	                            #ss_PLCIDTRAYID := CONCAT(IN1 := '0',
	                                                      IN2 := #ss_PLCIDTRAYID);

	                        END_FOR;

	                    END_IF;

	                    // PLCID/TRAYID addition
	                    #ss_PLCIDTRAYID := INSERT(IN1 := #ss_PLCIDTRAYID, IN2 := #is_PLCID_TRAYID, P := 0);

	                    // Delay preparation
	                    #ss_Delay := '';

	                    // Delay integer input conversion to a character string
	                    VAL_STRG(IN := #ii_Delay,
	                             SIZE := 0,
	                             PREC := 0,
	                             FORMAT := 0,
	                             P := 1,
	                             OUT => #ss_Delay);

	                    // Length of the delay character string
	                    #si_DelayLen := LEN(#ss_Delay);

	                    // Delay character string leading zeros addition
	                    IF (#si_DelayLen < 4)
	                    THEN

	                        FOR #si_i := 1 TO 4 - #si_DelayLen DO

	                            #ss_Delay := CONCAT(IN1 := '0',
	                                                IN2 := #ss_Delay);

	                        END_FOR;

	                    END_IF;

	                    // Message preparation

	                    // IDFWD message composing according to the structure: SCN,SCT,RCN,RCT,MT,MSGID,PLCID,DESSYS,DELAY{CRLF}
	                    #ss_Message := CONCAT(IN1 := #iUDT_MsgHeader.SCN,          // Sender IP address
	                                          IN2 := #cc_DL,                        // Comma sign - ","
	                                          IN3 := #iUDT_MsgHeader.SCT,          // Sender Name
	                                          IN4 := #cc_DL,                        // Comma sign - ","
	                                          IN5 := #iUDT_MsgHeader.RCN,          // Receiver IP address
	                                          IN6 := #cc_DL,                        // Comma sign - ","
	                                          IN7 := #iUDT_MsgHeader.RCT,          // Receiver Name
	                                          IN8 := #cc_DL,                        // Comma sign - ","
	                                          IN9 := #cs_IDFWD,                     // Message type - "IDFWD"
	                                          IN10 := #cc_DL,                       // Comma sign - ","
	                                          IN11 := #ss_MSGID,                    // MSGID
	                                          IN12 := #cc_DL,                       // Comma sign - ","
	                                          IN13 := #ss_PLCIDTRAYID,             // PLCID
	                                          IN14 := #cc_DL,                       // Comma sign - ","
	                                          IN15 := #ss_DesSys,                   // Designated system
	                                          IN16 := #cc_DL,                       // Comma sign - ","
	                                          IN17 := #ss_Delay,                    // Delay time
	                                          IN18 := #cs_CRLF);                    // Termination signs - "$R$L"

	                    // Maximum number of the message characters
	                    #si_MaxMsgLen := "FC_GetNrOfArrayEl"(iv_Array := #s_UDT_MessageArray.Character);

	                    // Length of the complete message
	                    #si_MsgLen := LEN(#ss_Message);

	                    // Message array size validation
	                    #ss_Status.InvalidMsgArraySize := #si_MsgLen > #si_MaxMsgLen;

	                    // Message character String conversion into the message array of characters
	                    IF (NOT #ss_Status.InvalidMsgArraySize)
	                    THEN

	                        Strg_TO_Chars(Strg := #ss_Message,
	                                      pChars := 0,
	                                      Cnt => #sui_MsgArrayElNr,
	                                      Chars := #s_UDT_MessageArray.Character);

	                    END_IF;

	                    // Clearing remaining characters in the message character array
	                    IF (NOT #ss_Status.InvalidMsgArraySize)
	                    THEN

	                        // Filling up not used message character array elements with '$00' (ASCII - 16#00)
	                        FILL_BLK(IN := #cc_NULL,
	                                 COUNT := UINT_TO_ULINT(INT_TO_UINT(#si_MaxMsgLen) - #sui_MsgArrayElNr),
	                                 OUT => #s_UDT_MessageArray.Character[#sui_MsgArrayElNr]);

	                    END_IF;

	                    // Message write into a FIFO register
	                    IF (NOT #ss_Status.InvalidMsgArraySize)
	                    THEN

	                        // Mode 'W' - Write FIFO record
	                        "FC_Fifo"(ic_Mode := 'W',
	                                  qUDT_Status => #ss_Status.FIFOStatus,
	                                  qx_Error => #ss_Status.FIFOError,
	                                  qx_Warning => #ss_Status.FIFOWarning,
	                                  iqv_Data := #s_UDT_MessageArray,
	                                  iqUDT_FifoHeader := #iqUDT_FifoHeader,
	                                  iqv_DataBuffer := #iqa_FifoData);

	                        // Message sent as a destination request
	                        "DB_GIN".GIN[#ii_GIN].General.DestReqSend := #ix_DestinationRequest;

	                    END_IF;

	                    // In case of FIFO full, the FIFO full error bit and FIFO collective error bit are set
	                ELSE

	                    #ss_Status.FIFOError := TRUE;
	                    #ss_Status.FIFOStatus.FifoFull := TRUE;

	                END_IF;

	            END_IF;

	        END_REGION

	        REGION 1.4 – Status

	            // Parametrization collective error output
	            #qx_Error :=
	            #ss_Status.InvalidDesSysPar
	            OR #ss_Status.InvalidDelay
	            OR #ss_Status.InvalidGIN
	            OR #ss_Status.InvalidMsgArraySize
	            OR #ss_Status.FIFOError;

	            // Parametrization collective warning output
	            #qx_Warning := #ss_Status.FIFOWarning;

	        END_REGION

	    END_IF;

	END_REGION
END_FUNCTION_BLOCK

FUNCTION_BLOCK "FB_UPSLogon"
TITLE = FB_Logon
{ S7_Optimized_Access := 'TRUE' }
AUTHOR : MHSE
FAMILY : UPS_SpecificCommunication
VERSION : 3.0
// ATTRIBUTES
// AUTO_NUMBER = True
// BLOCK_NUMBER = 57
// END_ATTRIBUTES
//Function block to prepare and send UPS LOGON and FILTER messages.
   VAR_INPUT
      iUDT_Connection { ExternalAccessible := 'False'; ExternalVisible := 'False'; ExternalWritable := 'False'} : "UDT_Connection";   // Connection parameters
      iUDT_MsgHeader { ExternalAccessible := 'False'; ExternalVisible := 'False'; ExternalWritable := 'False'} : "UDT_UPSMessageHeader";   // UPS message header
      ia_MsgType { ExternalAccessible := 'False'; ExternalVisible := 'False'; ExternalWritable := 'False'} : Array[0..34] of String;   // UPS message types
      ix_ConEstablished { ExternalAccessible := 'False'; ExternalVisible := 'False'; ExternalWritable := 'False'} : Bool;   // TCPIP Connection established
   END_VAR

   VAR_OUTPUT
      qx_LogonOk { ExternalAccessible := 'False'; ExternalVisible := 'False'; ExternalWritable := 'False'} : Bool;   // FILTER and LOGON messages sent
   END_VAR

   VAR
      sFB_TSEND {InstructionName := 'TSEND'; LibVersion := '4.0'; ExternalAccessible := 'False'; ExternalVisible := 'False'; ExternalWritable := 'False'; S7_SetPoint := 'False'} : TSEND;   // Siemens "TSEND" block - to send the data over TCPIP socket
      sR_TRIG_ConEstablished {InstructionName := 'R_TRIG'; LibVersion := '1.0'; ExternalAccessible := 'False'; ExternalVisible := 'False'; ExternalWritable := 'False'; S7_SetPoint := 'False'} : R_TRIG;   // Siemens "R_Trig" - to prepare the rising edge trigger on "ix_ConEstablished" signal
      sR_TRIG_SendTrigFilter {InstructionName := 'R_TRIG'; LibVersion := '1.0'; ExternalAccessible := 'False'; ExternalVisible := 'False'; ExternalWritable := 'False'; S7_SetPoint := 'False'} : R_TRIG;   // Siemens "R_Trig" - to prepare the Filter send trigger
      sR_TRIG_SendTrigLogon {InstructionName := 'R_TRIG'; LibVersion := '1.0'; ExternalAccessible := 'False'; ExternalVisible := 'False'; ExternalWritable := 'False'; S7_SetPoint := 'False'} : R_TRIG;   // Siemens "R_Trig" - to prepare the LOGON send trigger
      sa_TSEND { ExternalAccessible := 'False'; ExternalVisible := 'False'; ExternalWritable := 'False'} : Struct   // TSEND block parameter structure
         Status { ExternalAccessible := 'False'; ExternalVisible := 'False'; ExternalWritable := 'False'} : Word;
         Req { ExternalAccessible := 'False'; ExternalVisible := 'False'; ExternalWritable := 'False'} : Bool;
         Busy { ExternalAccessible := 'False'; ExternalVisible := 'False'; ExternalWritable := 'False'} : Bool;
         Done { ExternalAccessible := 'False'; ExternalVisible := 'False'; ExternalWritable := 'False'} : Bool;
         Error { ExternalAccessible := 'False'; ExternalVisible := 'False'; ExternalWritable := 'False'} : Bool;
      END_STRUCT;
      sa_FilterMsg { ExternalAccessible := 'False'; ExternalVisible := 'False'; ExternalWritable := 'False'} : Array[0..699] of Char;   // FILTER message character array
      sa_LogonMsg { ExternalAccessible := 'False'; ExternalVisible := 'False'; ExternalWritable := 'False'} : Array[0..34] of Char;   // LOGON message character array
      ss_Logon { ExternalAccessible := 'False'; ExternalVisible := 'False'; ExternalWritable := 'False'} : String;   // LOGON message character string
      ss_Header { ExternalAccessible := 'False'; ExternalVisible := 'False'; ExternalWritable := 'False'} : String;   // Message header character string
      ss_Filter_1 { ExternalAccessible := 'False'; ExternalVisible := 'False'; ExternalWritable := 'False'} : String;   // FILTER message part 1 character string
      ss_Filter_2 { ExternalAccessible := 'False'; ExternalVisible := 'False'; ExternalWritable := 'False'} : String;   // FILTER message part 2 character string
      ss_Footer { ExternalAccessible := 'False'; ExternalVisible := 'False'; ExternalWritable := 'False'} : String;   // FILTER message footer character string
      sui_ArrayOffset { ExternalAccessible := 'False'; ExternalVisible := 'False'; ExternalWritable := 'False'} : UInt;   // Offset for writing in the array
      sui_FilterArrayElNr { ExternalAccessible := 'False'; ExternalVisible := 'False'; ExternalWritable := 'False'} : UInt;   // Number of written FILTER characters
      sui_LogonArrayElNr { ExternalAccessible := 'False'; ExternalVisible := 'False'; ExternalWritable := 'False'} : UInt;   // Number of written LOGON characters
      si_MaxNrOfMsgTypes { ExternalAccessible := 'False'; ExternalVisible := 'False'; ExternalWritable := 'False'} : Int;   // Maximum number of message types
      si_MaxFilterLen { ExternalAccessible := 'False'; ExternalVisible := 'False'; ExternalWritable := 'False'} : Int;   // Maximum number of FILTER message characters
      si_MaxLogonLen { ExternalAccessible := 'False'; ExternalVisible := 'False'; ExternalWritable := 'False'} : Int;   // Maximum number of LOGON message characters
      si_i { ExternalAccessible := 'False'; ExternalVisible := 'False'; ExternalWritable := 'False'} : Int;   // Loop counter
      sx_LogProc { ExternalAccessible := 'False'; ExternalVisible := 'False'; ExternalWritable := 'False'} : Bool;   // Logon procedure
      sx_FilterSent { ExternalAccessible := 'False'; ExternalVisible := 'False'; ExternalWritable := 'False'} : Bool;   // FILTER message sent
      sx_LogonSent { ExternalAccessible := 'False'; ExternalVisible := 'False'; ExternalWritable := 'False'} : Bool;   // LOGON message sent
   END_VAR

   VAR CONSTANT
      cc_DL : Char := ',';   // Comma sign
      cs_Filter : String := 'FILTER';   // Message type
      cs_Logon : String := 'LOGON';   // Message type
      cs_Pipe : String := ',|,';   // FILTER message element - ,|,
      cs_MT : String := 'MT,$'';   // FILTER message element - MT,'
      cs_Q : String := '$',=';   // FILTER message element - ',=
      cs_CRLF : String := '$R$L';   // Termination signs
   END_VAR


BEGIN
	(*
	----------------------------------------------------------------------------------------

	Version history:
	Date        | Version   | Author        | Remark
	----------------------------------------------------------------------------------------
	24/05/2019  | 0.1       | L.Klar        | first release MHS TIA 15.1
	24/07/2019  | 2.0       | L.Klar        | 2.0 MHS library release TIA 15.1
	23/08/2019  | 2.1       | K.Pokorski    | Comments simplified
	12/11/2019  | 3.0       | P.Majka       | 3.0 MHS library release TIA 15.1
	22/02/2023  | 4.0       | F.Baten       | 4.0 Release TIA 17.5
	*)

	REGION 1 – Connection check

	    // TCIPI connection established rising edge
	    #sR_TRIG_ConEstablished(CLK := #ix_ConEstablished);

	    // Logon process start
	    IF (#sR_TRIG_ConEstablished.Q)                             // Connection established rising edge
	    THEN

	        #sx_LogProc := TRUE;

	    END_IF;

	    // Message send confirmation bits reset in case of connection lost
	    IF (NOT #ix_ConEstablished)                                 // Connection terminated
	    THEN

	        #sx_FilterSent := FALSE;
	        #sx_LogonSent := FALSE;

	    END_IF;

	END_REGION

	REGION 2 – Assembly FILTER message

	    IF (#sx_LogProc)                                            // Logon procedure
	    THEN

	        // Resetting all components of the "Filter" message
	        REGION 2.1 – Initialization

	            #si_i := 0;
	            #sui_ArrayOffset := 0;
	            #sui_FilterArrayElNr := 0;
	            #ss_Header := '';
	            #ss_Filter_1 := '';
	            #ss_Filter_2 := '';
	            #ss_Footer := '';

	        END_REGION

	        REGION 2.2 – Maximum number of the message types array elements

	            #si_MaxNrOfMsgTypes := "FC_GetNrOfArrayEl"(iv_Array := #ia_MsgType);

	        END_REGION

	        REGION 2.3 – Maximum number of the FILTER message array elements

	            #si_MaxFilterLen := "FC_GetNrOfArrayEl"(iv_Array := #sa_FilterMsg);

	        END_REGION

	        // Combining all components of the FILTER message header into one character string
	        REGION 2.4 – Assembly FILTER message header

	            #ss_Header := CONCAT(IN1 := #iUDT_MsgHeader.SCN,       // Sender IP address
	                                 IN2 := #cc_DL,                     // Comma sign - ","
	                                 IN3 := #iUDT_MsgHeader.SCT,       // Sender Name
	                                 IN4 := #cc_DL,                     // Comma sign - ","
	                                 IN5 := #cc_DL,                     // Comma sign - ","
	                                 IN6 := #cc_DL,                     // Comma sign - ","
	                                 IN7 := #cs_Filter,                 // Message type - "FILTER"
	                                 IN8 := #cc_DL);                    // Comma sign - ","

	        END_REGION


	        REGION 2.5 – Assembly FILTER message

	            // Combining all components of the FILTER message into one character string
	            FOR #si_i := 0 TO #si_MaxNrOfMsgTypes - 1 DO

	                IF (#ia_MsgType[#si_i] <> '')       // Message type isn't empty
	                THEN

	                    //  Message charater string conversion to a message array characters
	                    IF (#si_i = 0)                                                          // Loop counter equal to 0
	                    THEN

	                        #ss_Filter_1 := CONCAT(IN1 := #cs_MT,                               // FILTER message constant - "MT,'"
	                                               IN2 := #ia_MsgType[#si_i],                   // Used message type
	                                               IN3 := #cs_Q,                                // FILTER message constant - "',="
	                                               IN4 := #cc_DL);                              // Comma sign - ","

	                        // Message header character string into the character array conversion
	                        Strg_TO_Chars(Strg := #ss_Header,
	                                      pChars := 0,
	                                      Cnt => #sui_ArrayOffset,
	                                      Chars := #sa_FilterMsg);

	                        // FILTER message part 1 character string into the character array conversion
	                        Strg_TO_Chars(Strg := #ss_Filter_1,
	                                      pChars := #sui_ArrayOffset,
	                                      Cnt => #sui_FilterArrayElNr,
	                                      Chars := #sa_FilterMsg);

	                        // Handled message types addition to a filter message
	                    ELSIF (#si_i > 0)                                                       // Loop counter is greater than 0
	                    THEN

	                        #ss_Filter_2 := CONCAT(IN1 := #cs_MT,                               // FILTER message constant - "MT,'"
	                                               IN2 := #ia_MsgType[#si_i],                   // Used message type
	                                               IN3 := #cs_Q,                                // FILTER message constant - "',="
	                                               IN4 := #cs_Pipe);                            // FILTER message constant - ",|,"

	                        // Array offset update
	                        #sui_ArrayOffset += #sui_FilterArrayElNr;

	                        // FILTER message part 2 character string into the character array conversion
	                        Strg_TO_Chars(Strg := #ss_Filter_2,
	                                      pChars := #sui_ArrayOffset,
	                                      Cnt => #sui_FilterArrayElNr,
	                                      Chars := #sa_FilterMsg);

	                    END_IF;

	                    // The message type array element is empty
	                ELSE

	                    EXIT;

	                END_IF;

	            END_FOR;

	        END_REGION

	        REGION 2.6 – Assembly FILTER message footer

	            // FILTER footer creation
	            #ss_Footer := #cs_CRLF;

	            // Array offset update
	            #sui_ArrayOffset += #sui_FilterArrayElNr;

	            // FILTER footer character string into the character array conversion
	            Strg_TO_Chars(Strg := #ss_Footer,
	                          pChars := #sui_ArrayOffset,
	                          Cnt => #sui_FilterArrayElNr,
	                          Chars := #sa_FilterMsg);

	        END_REGION

	        REGION 2.7 – Clearing remaining characters in the message character array

	            // Filling up not used FILTER character array elements with '$00' (ASCII - 16#00)
	            FILL_BLK(IN := '$00',
	                     COUNT := UINT_TO_ULINT(INT_TO_UINT(#si_MaxFilterLen) -
	                                            #sui_FilterArrayElNr -
	                                            #sui_ArrayOffset),
	                     OUT => #sa_FilterMsg[#sui_ArrayOffset + #sui_FilterArrayElNr]);

	        END_REGION

	    END_IF;

	END_REGION

	REGION 3 – Assembly LOGON message

	    IF (#sx_LogProc)        // Logon procedure
	    THEN

	        REGION 3.1 – Initialization

	            #ss_Logon := '';

	        END_REGION

	        REGION 3.2 – Maximum number of the LOGON message array elements

	            #si_MaxLogonLen := "FC_GetNrOfArrayEl"(iv_Array := #sa_LogonMsg);

	        END_REGION

	        REGION 3.3 – Assembly LOGON message

	            #ss_Logon := CONCAT(IN1 := #iUDT_MsgHeader.SCN,        // Sender IP address
	                                IN2 := #cc_DL,                      // Comma sign - ","
	                                IN3 := #iUDT_MsgHeader.SCT,        // Sender Name
	                                IN4 := #cc_DL,                      // Comma sign - ","
	                                IN5 := #cc_DL,                      // Comma sign - ","
	                                IN6 := #cc_DL,                      // Comma sign - ","
	                                IN7 := #cs_Logon,                   // Message type - "LOGON"
	                                IN8 := #cs_CRLF);                   // Termination signs - "$R$L"

	            // LOGON message character string into the character array conversion
	            Strg_TO_Chars(Strg := #ss_Logon,
	                          pChars := 0,
	                          Cnt => #sui_LogonArrayElNr,
	                          Chars := #sa_LogonMsg);

	        END_REGION

	        REGION 3.4 – Clearing remaining characters in the message character array

	            // Filling up not used LOGON character array elements with '$00' (ASCII - 16#00)
	            FILL_BLK(IN := '$00',
	                     COUNT := UINT_TO_ULINT(INT_TO_UINT(#si_MaxLogonLen) -
	                                            #sui_LogonArrayElNr),
	                     OUT => #sa_LogonMsg[#sui_LogonArrayElNr]);

	        END_REGION

	    END_IF;

	END_REGION

	REGION 4 – Send FILTER message

	    REGION 4.1 – Send trigger preparation

	        #sR_TRIG_SendTrigFilter(CLK := NOT #sa_TSEND.#Busy
	                                AND #ix_ConEstablished
	                                AND #sx_LogProc
	                                AND NOT #sx_FilterSent
	                                AND NOT #sx_LogonSent,
	                                Q => #sa_TSEND.#Req);

	    END_REGION

	    REGION 4.2 – Send message

	        IF (NOT #sx_FilterSent               // FILTER message not sent
	            AND NOT #sx_LogonSent)           // LOGON message not sent
	        THEN

	            // FILTER message send
	            #sFB_TSEND(REQ := #sa_TSEND.#Req,
	                       ID := #iUDT_Connection.ID,
	                       LEN := #sui_ArrayOffset + #sui_FilterArrayElNr,
	                       DONE => #sa_TSEND.Done,
	                       BUSY => #sa_TSEND.Busy,
	                       ERROR => #sa_TSEND.Error,
	                       STATUS => #sa_TSEND.Status,
	                       DATA := #sa_FilterMsg);

	            // FILTER sent
	            IF (#sa_TSEND.#Done)        // Operation is done
	            THEN

	                #sx_FilterSent := TRUE;

	            END_IF;

	        END_IF;

	    END_REGION

	END_REGION

	REGION 5 – LOGON message send

	    REGION 5.1 – Send trigger preparation

	        #sR_TRIG_SendTrigLogon(CLK := NOT #sa_TSEND.Busy       // TSEND block not busy
	                               AND #ix_ConEstablished          // Connection established
	                               AND #sx_LogProc                 // Logon procedure
	                               AND #sx_FilterSent              // FILTER message is sent
	                               AND NOT #sx_LogonSent,          // LOGON message is not sent
	                               Q => #sa_TSEND.Req);

	    END_REGION

	    REGION 5.2 – Send message

	        IF (#sx_FilterSent              // FILTER mseesge is sent
	            AND NOT #sx_LogonSent)      // LOGON message is not sent
	        THEN
	            // LOGON message send
	            #sFB_TSEND(REQ := #sa_TSEND.#Req,
	                       ID := #iUDT_Connection.ID,
	                       LEN := #sui_LogonArrayElNr,
	                       DONE => #sa_TSEND.#Done,
	                       BUSY => #sa_TSEND.#Busy,
	                       ERROR => #sa_TSEND.#Error,
	                       STATUS => #sa_TSEND.#Status,
	                       DATA := #sa_LogonMsg);

	            // LOGON sent
	            IF (#sa_TSEND.#Done)        // Operation is done
	            THEN

	                #sx_LogonSent := TRUE;

	            END_IF;

	        END_IF;

	    END_REGION

	END_REGION

	REGION 6 – Reset Logon procedure

	    IF (#sx_FilterSent               // FILTER message sent
	        AND #sx_LogonSent)           // LOGON message sent
	    THEN

	        #sx_LogProc := FALSE;

	    END_IF;

	END_REGION

	REGION 7 – Write outputs

	    #qx_LogonOk :=
	    #sx_FilterSent            // FILTER message sent
	    AND #sx_LogonSent;        // LOGON message sent

	END_REGION
END_FUNCTION_BLOCK

FUNCTION_BLOCK "FB_UPSPLCInfo"
TITLE = FB_PLCInfo
{ S7_Optimized_Access := 'TRUE' }
AUTHOR : MHSE
FAMILY : UPS_SpecificCommunication
VERSION : 3.0
// ATTRIBUTES
// AUTO_NUMBER = True
// BLOCK_NUMBER = 58
// END_ATTRIBUTES
//Function block to prepare and send the UPS PLCINFO message.
   VAR_INPUT
      iUDT_MsgHeader { ExternalAccessible := 'False'; ExternalVisible := 'False'; ExternalWritable := 'False'} : "UDT_UPSMessageHeader";   // UPS message header
      iUDT_MachStat { ExternalAccessible := 'False'; ExternalVisible := 'False'; ExternalWritable := 'False'} : "UDT_UPSMACHSTAT";   // Machine status
      iUDT_ExternalReaders { ExternalAccessible := 'False'; ExternalVisible := 'False'; ExternalWritable := 'False'} : Array[0..15] of "UDT_UPSExternalReader";   // Active camera
      is_ActualDateTime { ExternalAccessible := 'False'; ExternalVisible := 'False'; ExternalWritable := 'False'} : String[23];   // Actual date and time
      is_ModuleName { ExternalAccessible := 'False'; ExternalVisible := 'False'; ExternalWritable := 'False'} : String[2] := 'AB';   // Module type
      is_DeviceNumber { ExternalAccessible := 'False'; ExternalVisible := 'False'; ExternalWritable := 'False'} : String[4] := 'abcd';   // Device number
      iudi_Speed { ExternalAccessible := 'False'; ExternalVisible := 'False'; ExternalWritable := 'False'} : UDInt;   // Conveyor speed [ft/min]
      iudi_SysRevs { ExternalAccessible := 'False'; ExternalVisible := 'False'; ExternalWritable := 'False'} : UDInt;   // Number of system revolutions since sort start
      ii_SendTimeInterval { ExternalAccessible := 'False'; ExternalVisible := 'False'; ExternalWritable := 'False'} : UInt;   // Send time interval [ms]
      ix_ExternalTrigger { ExternalAccessible := 'False'; ExternalVisible := 'False'; ExternalWritable := 'False'} : Bool;   // External trigger to send a message
   END_VAR

   VAR_OUTPUT
      qx_Error { ExternalAccessible := 'False'; ExternalVisible := 'False'; ExternalWritable := 'False'} : Bool;   // Collective error output
      qx_Warning { ExternalAccessible := 'False'; ExternalVisible := 'False'; ExternalWritable := 'False'} : Bool;   // Collective warning output
   END_VAR

   VAR_IN_OUT
      iqUDT_FifoHeader : "UDT_FifoHeader";   // FIFO header
      iqa_FifoData : Array[*] of "UDT_Message";   // FIFO data
      iqdi_UniqueMsgID { ExternalAccessible := 'False'; ExternalVisible := 'False'; ExternalWritable := 'False'} : DInt;   // Unique message ID integer
   END_VAR

   VAR
      sUDT_ActiveCamera { ExternalAccessible := 'False'; ExternalVisible := 'False'; ExternalWritable := 'False'; S7_SetPoint := 'False'} : Array[0..15] of "UDT_UPSExternalReader";   // Active camera status
      sa_MachStatArray { ExternalAccessible := 'False'; ExternalVisible := 'False'; ExternalWritable := 'False'} : Array[0..15] of Byte;   // Machine status array
      sR_TRIG_ExternaReq {InstructionName := 'R_TRIG'; LibVersion := '1.0'; ExternalAccessible := 'False'; ExternalVisible := 'False'; ExternalWritable := 'False'; S7_SetPoint := 'False'} : R_TRIG;   // Siemens "R_TRIG" - to prepare the rising edge trigger on "ix_ExternalTrigger" signal
      sF_TRIG_ExternalReq {InstructionName := 'F_TRIG'; LibVersion := '1.0'; ExternalAccessible := 'False'; ExternalVisible := 'False'; ExternalWritable := 'False'; S7_SetPoint := 'False'} : F_TRIG;   // Siemens "F_TRIG" - to prepare the falling edge trigger on "ix_ExternalTrigger" signal
      sFB_SendPulse { ExternalAccessible := 'False'; ExternalVisible := 'False'; ExternalWritable := 'False'; S7_SetPoint := 'False'} : "FB_Pulse";   // MHS "FB_Pulse" block - to generate preset pulse signal
      sUDT_MessageArray { ExternalAccessible := 'False'; ExternalVisible := 'False'; ExternalWritable := 'False'; S7_SetPoint := 'False'} : "UDT_Message";   // Message character array
      sa_Status { ExternalAccessible := 'False'; ExternalVisible := 'False'; ExternalWritable := 'False'} : Struct   // Status structure
         FIFOStatus { ExternalAccessible := 'False'; ExternalVisible := 'False'; ExternalWritable := 'False'} : "UDT_FifoStatus";   // FIFO status structure
         FIFOError { ExternalAccessible := 'False'; ExternalVisible := 'False'; ExternalWritable := 'False'; S7_SetPoint := 'True'} : Bool;   // FIFO error
         FIFOWarning { ExternalAccessible := 'False'; ExternalVisible := 'False'; ExternalWritable := 'False'; S7_SetPoint := 'True'} : Bool;   // FIFO warning
         InvalidSysRevs { ExternalAccessible := 'False'; ExternalVisible := 'False'; ExternalWritable := 'False'} : Bool;   // Invalid system revolutions number
         InvalidSpeed { ExternalAccessible := 'False'; ExternalVisible := 'False'; ExternalWritable := 'False'} : Bool;   // Invalid conveyor speed
         InvalidMsgArraySize { ExternalAccessible := 'False'; ExternalVisible := 'False'; ExternalWritable := 'False'} : Bool;   // Invalid message array size
      END_STRUCT;
      ss_MsgID { ExternalAccessible := 'False'; ExternalVisible := 'False'; ExternalWritable := 'False'} : String[32];   // Unique message ID
      ss_SysRevs { ExternalAccessible := 'False'; ExternalVisible := 'False'; ExternalWritable := 'False'} : String[4];   // Number of system revolutions since sort start
      ss_Speed { ExternalAccessible := 'False'; ExternalVisible := 'False'; ExternalWritable := 'False'} : String[5];   // Speed
      ss_CameraState { ExternalAccessible := 'False'; ExternalVisible := 'False'; ExternalWritable := 'False'} : String[2];   // Camera state character string
      ss_Header { ExternalAccessible := 'False'; ExternalVisible := 'False'; ExternalWritable := 'False'} : String;   // Header character string
      ss_Message { ExternalAccessible := 'False'; ExternalVisible := 'False'; ExternalWritable := 'False'} : String;   // Message character string
      ss_ActiveCamera { ExternalAccessible := 'False'; ExternalVisible := 'False'; ExternalWritable := 'False'} : String;   // Active camera character string
      ss_MachStat { ExternalAccessible := 'False'; ExternalVisible := 'False'; ExternalWritable := 'False'} : String;   // Machine status character string
      ss_MachStatPart { ExternalAccessible := 'False'; ExternalVisible := 'False'; ExternalWritable := 'False'} : String;   // Part of the machine status character string
      sui_MsgArrayElNr { ExternalAccessible := 'False'; ExternalVisible := 'False'; ExternalWritable := 'False'} : UInt;   // Number of written message characters
      sui_ArrayOffset { ExternalAccessible := 'False'; ExternalVisible := 'False'; ExternalWritable := 'False'} : UInt;   // Offset for writing in the array
      si_MaxMsgLen { ExternalAccessible := 'False'; ExternalVisible := 'False'; ExternalWritable := 'False'} : Int;   // Maximum message length
      si_MsgLen { ExternalAccessible := 'False'; ExternalVisible := 'False'; ExternalWritable := 'False'} : Int;   // Message character string length
      si_SysRevsLen { ExternalAccessible := 'False'; ExternalVisible := 'False'; ExternalWritable := 'False'} : Int;   // System revolutions character string length
      si_i { ExternalAccessible := 'False'; ExternalVisible := 'False'; ExternalWritable := 'False'} : Int;   // Loop counter
      sx_NewCameraState { ExternalAccessible := 'False'; ExternalVisible := 'False'; ExternalWritable := 'False'} : Bool;   // Camera state changed
   END_VAR

   VAR CONSTANT
      cc_NULL : Char := '$00';   // NULL sign
      cc_Dash : Char := '-';   // Dash sign
      cc_DL : Char := ',';   // Comma sign
      cs_CamOn : String := '|1';   // Camera state - True
      cs_CamOff : String := '|0';   // Camera state - False
      cs_PLCInfo : String := 'PLCINFO';   // Message type
      cs_CRLF : String := '$R$L';   // Termination signs
   END_VAR


BEGIN
	(*
	----------------------------------------------------------------------------------------

	Version history:
	Date        | Version   | Author        | Remark
	----------------------------------------------------------------------------------------
	24/05/2019  | 0.1       | L.Klar        | first release MHS TIA 15.1
	13/06/2019  | 0.2       | A.Nowak       | Replacement of instruction if for direct write into variable - Region 2 and 3 and 4.10
	28/06/2019  | 0.4       | A.Nowak       | Changing conditions for error occuring and status update
	18/07/2019  | 0.5       | L.Klar        | Status handling changed
	24/07/2019  | 2.0       | L.Klar        | 2.0 MHS library release TIA 15.1
	19/08/2019  | 2.1       | L.Klar        | Cyclic and event message handling added
	23/08/2019  | 2.2       | K.Pokorski    | Bool to byte block changed to direct reference, comments simplified
	20/09/2019  | 2.3       | M.Kurpiers    | Change - status to struct
	01/10/2019  | 2.4       | A.Nowak       | Implementation of the new FIFO block
	12/11/2019  | 3.0       | P.Majka       | 3.0 MHS library release TIA 15.1
	22/02/2023  | 4.0       | F.Baten       | 4.0 Release TIA 17.5
	02/05/2024  | 4.1       | J.Majer      | Datatype conversions changed from automatic to explicit, to accomodate IEC 61131-3 standard
	*)

	REGION 1 – Message send trigger

	    // Custom pulse to create cyclic trigger
	    #sFB_SendPulse(iudi_PulseTime := #ii_SendTimeInterval);

	    // Camera state check
	    #sx_NewCameraState := #sUDT_ActiveCamera <> #iUDT_ExternalReaders;
	    #sUDT_ActiveCamera := #iUDT_ExternalReaders;                             // Move new camera state to block memory

	    // Preparation of the rising and falling edge on the external request to send signal
	    #sR_TRIG_ExternaReq(CLK := #ix_ExternalTrigger);
	    #sF_TRIG_ExternalReq(CLK := #ix_ExternalTrigger);

	END_REGION

	REGION 2 – PLCInfo message request

	    // Condition of sending the message
	    IF (#sFB_SendPulse.qx_Pulse                // Cyclic trigger
	        OR #sx_NewCameraState                   // Camera state changed
	        OR #sR_TRIG_ExternaReq.Q               // External trigger rising edge
	        OR #sF_TRIG_ExternalReq.Q)             // External trigger falling edge
	    THEN

	        REGION 2.1 – FIFO header status update

	            // Mode 'S' - FIFO register status update
	            "FC_Fifo"(ic_Mode := 'S',
	                      qUDT_Status => #sa_Status.FIFOStatus,
	                      qx_Error => #sa_Status.FIFOError,
	                      qx_Warning => #sa_Status.FIFOWarning,
	                      iqv_Data := #sUDT_MessageArray,
	                      iqUDT_FifoHeader := #iqUDT_FifoHeader,
	                      iqv_DataBuffer := #iqa_FifoData);


	        END_REGION

	        REGION 2.2 – Conveyor speed validation

	            #sa_Status.InvalidSpeed :=
	            #iudi_Speed < 0
	            OR #iudi_Speed > 99999;

	        END_REGION

	        REGION 2.3 – System revolutions number validation

	            #sa_Status.InvalidSysRevs :=
	            #iudi_SysRevs < 0
	            OR #iudi_SysRevs > 9999;

	        END_REGION

	        REGION 2.4 – PLCINFO message preparation

	            IF (NOT #sa_Status.InvalidSysRevs                                // System revolutions number is valid
	                AND NOT #sa_Status.InvalidSpeed                              // Conveyor speed is valid
	                AND NOT #sa_Status.FIFOError)                                // No FIFO errors
	            THEN

	                IF (NOT #iqUDT_FifoHeader.Status.Full)                      // FIFO isn't full
	                THEN

	                    // Unique MSGID
	                    "FC_UPSMsgId"(is_ActualDateTime := #is_ActualDateTime,
	                                  is_ModuleName := #is_ModuleName,
	                                  is_DeviceNumber := #is_DeviceNumber,
	                                  iqs_MSGID := #ss_MsgID,
	                                  iqdi_UniqueMsgID := #iqdi_UniqueMsgID);


	                    // Conveyor speed conversion
	                    VAL_STRG(IN := #iudi_Speed,
	                             SIZE := 0,
	                             PREC := 0,
	                             FORMAT := 0,
	                             P := 1,
	                             OUT => #ss_Speed);

	                    // Machine status conversion
	                    #sa_MachStatArray[0].%X0 := #iUDT_MachStat."OpsNormal".StopMCP;                     // MCP Stop PB          // Byte 1, Bit 0 - Operator Stop MCP Panel
	                    #sa_MachStatArray[0].%X1 := #iUDT_MachStat."OpsNormal".StopRemoteCon1;              // SSP         // Byte 1, Bit 1 - Operator Stop Remote Console 1
	                    #sa_MachStatArray[0].%X2 := #iUDT_MachStat."OpsNormal".StopRemoteCon2;              // SSP         // Byte 1, Bit 2 - Operator Stop Remote Console 2
	                    #sa_MachStatArray[0].%X3 := #iUDT_MachStat."OpsNormal".BuildingStop;                // MCP Estop         // Byte 1, Bit 3 - Building Stop via HMI
	                    #sa_MachStatArray[0].%X4 := #iUDT_MachStat."OpsNormal".BuildingBreak;               // false         // Byte 1, Bit 4 - Building Break Time via HMI
	                    #sa_MachStatArray[0].%X5 := #iUDT_MachStat."OpsNormal".PowerSaveShutdown;           // system energy save       // Byte 1, Bit 5 - Power Save Shutdown
	                    #sa_MachStatArray[0].%X6 := #iUDT_MachStat."OpsNormal".SorterNotAtSpeed;            //False        // Byte 1, Bit 6 - Sorter Not at speed
	                    #sa_MachStatArray[0].%X7 := #iUDT_MachStat."OpsNormal".MaintenanceSysMode;          // Manual      // Byte 1, Bit 7 - System in Maintenance Mode

	                    #sa_MachStatArray[1].%X0 := #iUDT_MachStat."OpsNormal".Spare_8;                     // Byte 2, Bit 0 - Future / or Machine Specific (To be identified)
	                    #sa_MachStatArray[1].%X1 := #iUDT_MachStat."OpsNormal".Spare_9;                     // Byte 2, Bit 1 - Future / or Machine Specific (To be identified)
	                    #sa_MachStatArray[1].%X2 := #iUDT_MachStat."OpsNormal".Spare_10;                    // Byte 2, Bit 2 - Future / or Machine Specific (To be identified)
	                    #sa_MachStatArray[1].%X3 := #iUDT_MachStat."OpsNormal".Spare_11;                    // Byte 2, Bit 3 - Future / or Machine Specific (To be identified)
	                    #sa_MachStatArray[1].%X4 := #iUDT_MachStat."OpsNormal".Spare_12;                    // Byte 2, Bit 4 - Future / or Machine Specific (To be identified)
	                    #sa_MachStatArray[1].%X5 := #iUDT_MachStat."OpsNormal".Spare_13;                    // Byte 2, Bit 5 - Future / or Machine Specific (To be identified)
	                    #sa_MachStatArray[1].%X6 := #iUDT_MachStat."OpsNormal".Spare_14;                    // Byte 2, Bit 6 - Future / or Machine Specific (To be identified)
	                    #sa_MachStatArray[1].%X7 := #iUDT_MachStat."OpsNormal".Spare_15;                    // Byte 2, Bit 7 - Future / or Machine Specific (To be identified)


	                    #sa_MachStatArray[2].%X0 := #iUDT_MachStat."OpsNormal".Spare_16;                    // Byte 3, Bit 0 - Future / or Machine Specific (To be identified)
	                    #sa_MachStatArray[2].%X1 := #iUDT_MachStat."OpsNormal".Spare_17;                    // Byte 3, Bit 1 - Future / or Machine Specific (To be identified)
	                    #sa_MachStatArray[2].%X2 := #iUDT_MachStat."OpsNormal".Spare_18;                    // Byte 3, Bit 2 - Future / or Machine Specific (To be identified)
	                    #sa_MachStatArray[2].%X3 := #iUDT_MachStat."OpsNormal".Spare_19;                    // Byte 3, Bit 3 - Future / or Machine Specific (To be identified)
	                    #sa_MachStatArray[2].%X4 := #iUDT_MachStat."OpsNormal".Spare_20;                    // Byte 3, Bit 4 - Future / or Machine Specific (To be identified)
	                    #sa_MachStatArray[2].%X5 := #iUDT_MachStat."OpsNormal".Spare_21;                    // Byte 3, Bit 5 - Future / or Machine Specific (To be identified)
	                    #sa_MachStatArray[2].%X6 := #iUDT_MachStat."OpsNormal".Spare_22;                    // Byte 3, Bit 6 - Future / or Machine Specific (To be identified)
	                    #sa_MachStatArray[2].%X7 := #iUDT_MachStat."OpsNormal".Spare_23;                    // Byte 3, Bit 7 - Future / or Machine Specific (To be identified)


	                    #sa_MachStatArray[3].%X0 := #iUDT_MachStat."OpsNormal".Spare_24;                    // Byte 4, Bit 0 - Future / or Machine Specific (To be identified)
	                    #sa_MachStatArray[3].%X1 := #iUDT_MachStat."OpsNormal".Spare_25;                    // Byte 4, Bit 1 - Future / or Machine Specific (To be identified)
	                    #sa_MachStatArray[3].%X2 := #iUDT_MachStat."OpsNormal".Spare_26;                    // Byte 4, Bit 2 - Future / or Machine Specific (To be identified)
	                    #sa_MachStatArray[3].%X3 := #iUDT_MachStat."OpsNormal".Spare_27;                    // Byte 4, Bit 3 - Future / or Machine Specific (To be identified)
	                    #sa_MachStatArray[3].%X4 := #iUDT_MachStat."OpsNormal".Spare_28;                    // Byte 4, Bit 4 - Future / or Machine Specific (To be identified)
	                    #sa_MachStatArray[3].%X5 := #iUDT_MachStat."OpsNormal".Spare_29;                    // Byte 4, Bit 5 - Future / or Machine Specific (To be identified)
	                    #sa_MachStatArray[3].%X6 := #iUDT_MachStat."OpsNormal".Spare_30;                    // Byte 4, Bit 6 - Future / or Machine Specific (To be identified)
	                    #sa_MachStatArray[3].%X7 := #iUDT_MachStat."OpsNormal".Spare_31;                    // Byte 4, Bit 7 - Future / or Machine Specific (To be identified)


	                    #sa_MachStatArray[4].%X0 := #iUDT_MachStat.SafetyFaults.BuildingEStop;              // comm false           // Byte 5, Bit 0 - Building Emergency Stop
	                    #sa_MachStatArray[4].%X1 := #iUDT_MachStat.SafetyFaults.SystemEStop;                // MCP Estop          // Byte 5, Bit 1 - System Emergency Stop
	                    #sa_MachStatArray[4].%X2 := #iUDT_MachStat.SafetyFaults.EmerPullCord;               // Byte 5, Bit 2 - Emergency Pull Cord
	                    #sa_MachStatArray[4].%X3 := #iUDT_MachStat.SafetyFaults.PhotoEyeBlock1;             // Byte 5, Bit 3 - Safety Photo Eye Blocked (Long Range Photo Eye) 1
	                    #sa_MachStatArray[4].%X4 := #iUDT_MachStat.SafetyFaults.PlatformLockout1;           // Byte 5, Bit 4 - Platform Lockout 1
	                    #sa_MachStatArray[4].%X5 := #iUDT_MachStat.SafetyFaults.PlatformLockout2;           // Byte 5, Bit 5 - Platform Lockout 2
	                    #sa_MachStatArray[4].%X6 := #iUDT_MachStat.SafetyFaults.PhotoEyeBlock2;             // Byte 5, Bit 6 - Safety Photo Eye Blocked (Long Range Photo Eye) 2
	                    #sa_MachStatArray[4].%X7 := #iUDT_MachStat.SafetyFaults.PhotoEyeBlock3;             // Byte 5, Bit 7 - Safety Photo Eye Blocked (Long Range Photo Eye) 3


	                    #sa_MachStatArray[5].%X0 := #iUDT_MachStat.SafetyFaults.Spare_8;                    // Byte 6, Bit 0 - Future / or Machine Specific (To be identified)
	                    #sa_MachStatArray[5].%X1 := #iUDT_MachStat.SafetyFaults.Spare_9;                    // Byte 6, Bit 1 - Future / OR Machine Specific (TO be identified)
	                    #sa_MachStatArray[5].%X2 := #iUDT_MachStat.SafetyFaults.Spare_10;                   // Byte 6, Bit 2 - Future / or Machine Specific (To be identified)
	                    #sa_MachStatArray[5].%X3 := #iUDT_MachStat.SafetyFaults.Spare_11;                   // Byte 6, Bit 3 - Future / or Machine Specific (To be identified)
	                    #sa_MachStatArray[5].%X4 := #iUDT_MachStat.SafetyFaults.Spare_12;                   // Byte 6, Bit 4 - Future / or Machine Specific (To be identified)
	                    #sa_MachStatArray[5].%X5 := #iUDT_MachStat.SafetyFaults.Spare_13;                   // Byte 6, Bit 5 - Future / or Machine Specific (To be identified)
	                    #sa_MachStatArray[5].%X6 := #iUDT_MachStat.SafetyFaults.Spare_14;                   // Byte 6, Bit 6 - Future / or Machine Specific (To be identified)
	                    #sa_MachStatArray[5].%X7 := #iUDT_MachStat.SafetyFaults.Spare_15;                   // Byte 6, Bit 7 - Future / or Machine Specific (To be identified)


	                    #sa_MachStatArray[6].%X0 := #iUDT_MachStat.SafetyFaults.Spare_16;                   // Byte 7, Bit 0 - Future / or Machine Specific (To be identified)
	                    #sa_MachStatArray[6].%X1 := #iUDT_MachStat.SafetyFaults.Spare_17;                   // Byte 7, Bit 1 - Future / or Machine Specific (To be identified)
	                    #sa_MachStatArray[6].%X2 := #iUDT_MachStat.SafetyFaults.Spare_18;                   // Byte 7, Bit 2 - Future / or Machine Specific (To be identified)
	                    #sa_MachStatArray[6].%X3 := #iUDT_MachStat.SafetyFaults.Spare_19;                   // Byte 7, Bit 3 - Future / or Machine Specific (To be identified)
	                    #sa_MachStatArray[6].%X4 := #iUDT_MachStat.SafetyFaults.Spare_20;                   // Byte 7, Bit 4 - Future / or Machine Specific (To be identified)
	                    #sa_MachStatArray[6].%X5 := #iUDT_MachStat.SafetyFaults.Spare_21;                   // Byte 7, Bit 5 - Future / or Machine Specific (To be identified)
	                    #sa_MachStatArray[6].%X6 := #iUDT_MachStat.SafetyFaults.Spare_22;                   // Byte 7, Bit 6 - Future / or Machine Specific (To be identified)
	                    #sa_MachStatArray[6].%X7 := #iUDT_MachStat.SafetyFaults.Spare_23;                   // Byte 7, Bit 7 - Future / or Machine Specific (To be identified)


	                    #sa_MachStatArray[7].%X0 := #iUDT_MachStat.SafetyFaults.Spare_24;                   // Byte 8, Bit 0 - Future / or Machine Specific (To be identified)
	                    #sa_MachStatArray[7].%X1 := #iUDT_MachStat.SafetyFaults.Spare_25;                   // Byte 8, Bit 1 - Future / or Machine Specific (To be identified)
	                    #sa_MachStatArray[7].%X2 := #iUDT_MachStat.SafetyFaults.Spare_26;                   // Byte 8, Bit 2 - Future / or Machine Specific (To be identified)
	                    #sa_MachStatArray[7].%X3 := #iUDT_MachStat.SafetyFaults.Spare_27;                   // Byte 8, Bit 3 - Future / or Machine Specific (To be identified)
	                    #sa_MachStatArray[7].%X4 := #iUDT_MachStat.SafetyFaults.Spare_28;                   // Byte 8, Bit 4 - Future / or Machine Specific (To be identified)
	                    #sa_MachStatArray[7].%X5 := #iUDT_MachStat.SafetyFaults.Spare_29;                   // Byte 8, Bit 5 - Future / or Machine Specific (To be identified)
	                    #sa_MachStatArray[7].%X6 := #iUDT_MachStat.SafetyFaults.Spare_30;                   // Byte 8, Bit 6 - Future / or Machine Specific (To be identified)
	                    #sa_MachStatArray[7].%X7 := #iUDT_MachStat.SafetyFaults.Spare_31;                   // Byte 8, Bit 7 - Future / or Machine Specific (To be identified)


	                    #sa_MachStatArray[8].%X0 := #iUDT_MachStat.SystemFaults.PLCRackFault;               // RIO Error     // Byte 9, Bit 0 - PLC Rack Fault
	                    #sa_MachStatArray[8].%X1 := #iUDT_MachStat.SystemFaults.EncoderFault;               // Byte 9, Bit 1 - Encoder Fault
	                    #sa_MachStatArray[8].%X2 := #iUDT_MachStat.SystemFaults.TipperOrDiverterFault;      // Byte 9, Bit 2 - Tipper / Diverter Fault
	                    #sa_MachStatArray[8].%X3 := #iUDT_MachStat.SystemFaults.TCPConFail;                 // Byte 9, Bit 3 - TCP Connection Failure
	                    #sa_MachStatArray[8].%X4 := #iUDT_MachStat.SystemFaults.SensorJam;                  // Byte 9, Bit 4 - Package Detect Sensor Jam
	                    #sa_MachStatArray[8].%X5 := #iUDT_MachStat.SystemFaults.CamOrScanFail;              // health        // Byte 9, Bit 5 - Camera / Scanner Failure
	                    #sa_MachStatArray[8].%X6 := #iUDT_MachStat.SystemFaults.InductPEJam;                // Byte 9, Bit 6 - Induct Photo Eye Jam
	                    #sa_MachStatArray[8].%X7 := #iUDT_MachStat.SystemFaults.SortVerificationPEJam;      // Byte 9, Bit 7 - Sort Verification Photo Eye Jam


	                    #sa_MachStatArray[9].%X0 := #iUDT_MachStat.SystemFaults.TakeAwayConvPEJam;          // Byte 10, Bit 0 - Take Away Conveyor Photo Eye Jam
	                    #sa_MachStatArray[9].%X1 := #iUDT_MachStat.SystemFaults.SorterMechFault;            // Byte 10, Bit 1 - Sorter Mechanical Fault
	                    #sa_MachStatArray[9].%X2 := #iUDT_MachStat.SystemFaults.Spare_10;                   // Byte 10, Bit 2 - Future / or Machine Specific (To be identified)
	                    #sa_MachStatArray[9].%X3 := #iUDT_MachStat.SystemFaults.SorterJam;                  // Byte 10, Bit 3 - Sorter Jam (Logical Failure)
	                    #sa_MachStatArray[9].%X4 := #iUDT_MachStat.SystemFaults.InductPCAlignmentError;     // Byte 10, Bit 4 - Induct Photo Cell Alignment Error
	                    #sa_MachStatArray[9].%X5 := #iUDT_MachStat.SystemFaults.MotorFault;                 // Byte 10, Bit 5 - Motor Fault
	                    #sa_MachStatArray[9].%X6 := #iUDT_MachStat.SystemFaults.PowerFault;                 // PDP                // Byte 10, Bit 6 - Power Fault
	                    #sa_MachStatArray[9].%X7 := #iUDT_MachStat.SystemFaults.Spare_15;                   // Byte 10, Bit 7 - Future / or Machine Specific (To be identified)


	                    #sa_MachStatArray[10].%X0 := #iUDT_MachStat.SystemFaults.IOComError;                // Byte 11, Bit 0 - I/O Communications Error
	                    #sa_MachStatArray[10].%X1 := #iUDT_MachStat.SystemFaults.RemoteIOComError;          // Byte 11, Bit 1 - Remote I/O Communications Error
	                    #sa_MachStatArray[10].%X2 := #iUDT_MachStat.SystemFaults.XLeChatComError;           // Byte 11, Bit 2 - XLe chat Communications Error
	                    #sa_MachStatArray[10].%X3 := #iUDT_MachStat.SystemFaults.SerialComError;            // Byte 11, Bit 3 - Serial Communications Error
	                    #sa_MachStatArray[10].%X4 := #iUDT_MachStat.SystemFaults.SubsystemError;            // camera error           // Byte 11, Bit 4 - Subsystem Error (Scale, Camera, etc…)
	                    #sa_MachStatArray[10].%X5 := #iUDT_MachStat.SystemFaults.VDFFault;                  // Byte 11, Bit 5 - VDF Fault
	                    #sa_MachStatArray[10].%X6 := #iUDT_MachStat.SystemFaults.SystemResetInitiated;      // Byte 11, Bit 6 - System Reset Initiated
	                    #sa_MachStatArray[10].%X7 := #iUDT_MachStat.SystemFaults.PFCStopMode;               // Byte 11, Bit 7 - PFC not in Run Mode


	                    #sa_MachStatArray[11].%X0 := #iUDT_MachStat.SystemFaults.NoHitPoints;               // Byte 12, Bit 0 - No Hit points / Divert Set Points found
	                    #sa_MachStatArray[11].%X1 := #iUDT_MachStat.SystemFaults.MissingTraysDetected;      // Byte 12, Bit 1 - Missing Trays Detected
	                    #sa_MachStatArray[11].%X2 := #iUDT_MachStat.SystemFaults.DataFault;                 // Byte 12, Bit 2 - Data Fault, X number of sequential missing valid SORT messages
	                    #sa_MachStatArray[11].%X3 := #iUDT_MachStat.SystemFaults.Spare_27;                  // Byte 12, Bit 3 - Future / or Machine Specific (To be identified)
	                    #sa_MachStatArray[11].%X4 := #iUDT_MachStat.SystemFaults.Spare_28;                  // Byte 12, Bit 4 - Future / or Machine Specific (To be identified)
	                    #sa_MachStatArray[11].%X5 := #iUDT_MachStat.SystemFaults.Spare_29;                  // Byte 12, Bit 5 - Future / or Machine Specific (To be identified)
	                    #sa_MachStatArray[11].%X6 := #iUDT_MachStat.SystemFaults.Spare_30;                  // Byte 12, Bit 6 - Future / or Machine Specific (To be identified)
	                    #sa_MachStatArray[11].%X7 := #iUDT_MachStat.SystemFaults.Spare_31;                  // Byte 12, Bit 7 - Future / or Machine Specific (To be identified)


	                    #sa_MachStatArray[12].%X0 := #iUDT_MachStat.OtherFaults.ConsoleDisconnect;          // Byte 13, Bit 0 - Console Disconnect
	                    #sa_MachStatArray[12].%X1 := #iUDT_MachStat.OtherFaults.PLCChassisPower;            // Byte 13, Bit 1 - PLC Chassis Power
	                    #sa_MachStatArray[12].%X2 := #iUDT_MachStat.OtherFaults.SystemInputPower;           // Byte 13, Bit 2 - System Input Power
	                    #sa_MachStatArray[12].%X3 := #iUDT_MachStat.OtherFaults.SystemPowerOutput;          // Byte 13, Bit 3 - System Output Power
	                    #sa_MachStatArray[12].%X4 := #iUDT_MachStat.OtherFaults.DiverterTipperPower;        // Byte 13, Bit 4 - Diverter / Tipper Power
	                    #sa_MachStatArray[12].%X5 := #iUDT_MachStat.OtherFaults.VFDServoFault;              // Byte 13, Bit 5 - VFD / Servo Fault
	                    #sa_MachStatArray[12].%X6 := #iUDT_MachStat.OtherFaults.MotorStarterFault;          // Byte 13, Bit 6 - Motor Starter Fault
	                    #sa_MachStatArray[12].%X7 := #iUDT_MachStat.OtherFaults.PLCFault;                   // Byte 13, Bit 7 - PLC Fault


	                    #sa_MachStatArray[13].%X0 := #iUDT_MachStat.OtherFaults.Spare_8;                    // Byte 14, Bit 0 - Future / or Machine Specific (To be identified)
	                    #sa_MachStatArray[13].%X1 := #iUDT_MachStat.OtherFaults.Spare_9;                    // Byte 14, Bit 1 - Future / or Machine Specific (To be identified)
	                    #sa_MachStatArray[13].%X2 := #iUDT_MachStat.OtherFaults.Spare_10;                   // Byte 14, Bit 2 - Future / or Machine Specific (To be identified)
	                    #sa_MachStatArray[13].%X3 := #iUDT_MachStat.OtherFaults.Spare_11;                   // Byte 14, Bit 3 - Future / or Machine Specific (To be identified)
	                    #sa_MachStatArray[13].%X4 := #iUDT_MachStat.OtherFaults.Spare_12;                   // Byte 14, Bit 4 - Future / or Machine Specific (To be identified)
	                    #sa_MachStatArray[13].%X5 := #iUDT_MachStat.OtherFaults.Spare_13;                   // Byte 14, Bit 5 - Future / or Machine Specific (To be identified)
	                    #sa_MachStatArray[13].%X6 := #iUDT_MachStat.OtherFaults.Spare_14;                   // Byte 14, Bit 6 - Future / or Machine Specific (To be identified)
	                    #sa_MachStatArray[13].%X7 := #iUDT_MachStat.OtherFaults.Spare_15;                   // Byte 14, Bit 7 - Future / or Machine Specific (To be identified)


	                    #sa_MachStatArray[14].%X0 := #iUDT_MachStat.OtherFaults.Spare_16;                   // Byte 15, Bit 0 - Future / or Machine Specific (To be identified)
	                    #sa_MachStatArray[14].%X1 := #iUDT_MachStat.OtherFaults.Spare_17;                   // Byte 15, Bit 1 - Future / or Machine Specific (To be identified)
	                    #sa_MachStatArray[14].%X2 := #iUDT_MachStat.OtherFaults.Spare_18;                   // Byte 15, Bit 2 - Future / or Machine Specific (To be identified)
	                    #sa_MachStatArray[14].%X3 := #iUDT_MachStat.OtherFaults.Spare_19;                   // Byte 15, Bit 3 - Future / or Machine Specific (To be identified)
	                    #sa_MachStatArray[14].%X4 := #iUDT_MachStat.OtherFaults.Spare_20;                   // Byte 15, Bit 4 - Future / or Machine Specific (To be identified)
	                    #sa_MachStatArray[14].%X5 := #iUDT_MachStat.OtherFaults.Spare_21;                   // Byte 15, Bit 5 - Future / or Machine Specific (To be identified)
	                    #sa_MachStatArray[14].%X6 := #iUDT_MachStat.OtherFaults.Spare_22;                   // Byte 15, Bit 6 - Future / or Machine Specific (To be identified)
	                    #sa_MachStatArray[14].%X7 := #iUDT_MachStat.OtherFaults.Spare_23;                   // Byte 15, Bit 7 - Future / or Machine Specific (To be identified)


	                    #sa_MachStatArray[15].%X0 := #iUDT_MachStat.OtherFaults.Spare_24;                   // Byte 16, Bit 0 - Future / or Machine Specific (To be identified)
	                    #sa_MachStatArray[15].%X1 := #iUDT_MachStat.OtherFaults.Spare_25;                   // Byte 16, Bit 1 - Future / or Machine Specific (To be identified)
	                    #sa_MachStatArray[15].%X2 := #iUDT_MachStat.OtherFaults.Spare_26;                   // Byte 16, Bit 2 - Future / or Machine Specific (To be identified)
	                    #sa_MachStatArray[15].%X3 := #iUDT_MachStat.OtherFaults.Spare_27;                   // Byte 16, Bit 3 - Future / or Machine Specific (To be identified)
	                    #sa_MachStatArray[15].%X4 := #iUDT_MachStat.OtherFaults.Spare_28;                   // Byte 16, Bit 4 - Future / or Machine Specific (To be identified)
	                    #sa_MachStatArray[15].%X5 := #iUDT_MachStat.OtherFaults.Spare_29;                   // Byte 16, Bit 5 - Future / or Machine Specific (To be identified)
	                    #sa_MachStatArray[15].%X6 := #iUDT_MachStat.OtherFaults.Spare_30;                   // Byte 16, Bit 6 - Future / or Machine Specific (To be identified)
	                    #sa_MachStatArray[15].%X7 := #iUDT_MachStat.OtherFaults.Spare_31;                   // Byte 16, Bit 7 - Future / or Machine Specific (To be identified)


	                    // Machine status character string clearing
	                    #ss_MachStat := '';

	                    // Machine status bytes conversion to character string
	                    FOR #si_i := 0 TO 15 DO

	                        #ss_MachStatPart := '';                                                         // Machine status part of the character string clearing

	                        VAL_STRG(IN := BYTE_TO_USINT(#sa_MachStatArray[#si_i]),                                        // Machine status byte conversion to string
	                                 SIZE := 0,
	                                 PREC := 0,
	                                 FORMAT := 0,
	                                 P := 1,
	                                 OUT => #ss_MachStatPart);

	                        // MACHSTAT character string building
	                        IF (#si_i < 15)                                                                 // Loop counter lower than 15
	                        THEN

	                            #ss_MachStat := CONCAT(IN1 := #ss_MachStat,
	                                                   IN2 := #ss_MachStatPart,
	                                                   IN3 := #cc_Dash);

	                        ELSE

	                            #ss_MachStat := CONCAT(IN1 := #ss_MachStat,
	                                                   IN2 := #ss_MachStatPart);

	                        END_IF;

	                    END_FOR;

	                    // System revolutions number preparation

	                    // System revolutions number character string clearing
	                    #ss_SysRevs := '';

	                    // System revolutions number integer input conversion to a character string
	                    VAL_STRG(IN := #iudi_SysRevs,
	                             SIZE := 0,
	                             PREC := 0,
	                             FORMAT := 0,
	                             P := 1,
	                             OUT => #ss_SysRevs);

	                    // Length of the system revolutions number character string
	                    #si_SysRevsLen := LEN(#ss_SysRevs);

	                    // System revolutions number character string leading zeros addition
	                    IF (#si_SysRevsLen < 4)             // System revolutions character string length lower than 4
	                    THEN

	                        FOR #si_i := 1 TO 4 - #si_SysRevsLen DO

	                            #ss_SysRevs := CONCAT(IN1 := '0',
	                                                  IN2 := #ss_SysRevs);

	                        END_FOR;

	                    END_IF;

	                    // Active cameras

	                    // Active cameras character string clearing
	                    #ss_ActiveCamera := '';


	                    // Active cameras character string building
	                    // If the IP address of the camera is not empty, the proper string with its state is prepared.
	                    FOR #si_i := 0 TO 9 DO

	                        IF (#iUDT_ExternalReaders[#si_i].IPAddress <> '')      // Camera adres isn't empty
	                        THEN

	                            IF (#iUDT_ExternalReaders[#si_i].State)            // State on true
	                            THEN

	                                #ss_CameraState := #cs_CamOn;

	                            ELSE

	                                #ss_CameraState := #cs_CamOff;

	                            END_IF;

	                            IF (#si_i = 0)          // Loop counter equal to 0
	                            THEN

	                                #ss_ActiveCamera := CONCAT(IN1 := #ss_ActiveCamera,                                 // Active camera
	                                                           IN2 := #iUDT_ExternalReaders[#si_i].IPAddress,           // Camera IP address
	                                                           IN3 := #ss_CameraState);                                 // Camera state

	                            ELSE

	                                #ss_ActiveCamera := CONCAT(IN1 := #ss_ActiveCamera,                                 // Active camera
	                                                           IN2 := #cc_Dash,                                         // Dash sign - "-"
	                                                           IN3 := #iUDT_ExternalReaders[#si_i].IPAddress,           // Camera IP address
	                                                           IN4 := #ss_CameraState);                                 // Camera state

	                            END_IF;

	                        END_IF;

	                    END_FOR;

	                    // PLCINFO message composing according to the structure: SCN,SCT,RCN,RCT,MT,MSGID,SPEED,MACHSTAT,SYSREVS,ACTIVECAMERA {CRLF}
	                    #ss_Header := CONCAT(IN1 := #iUDT_MsgHeader.SCN,        // Sender IP address
	                                         IN2 := #cc_DL,                     // Comma sign - ","
	                                         IN3 := #iUDT_MsgHeader.SCT,        // Sender Name
	                                         IN4 := #cc_DL,                     // Comma sign - ","
	                                         IN5 := #iUDT_MsgHeader.RCN,        // Receiver IP address
	                                         IN6 := #cc_DL,                     // Comma sign - ","
	                                         IN7 := #iUDT_MsgHeader.RCT,        // Receiver Name
	                                         IN8 := #cc_DL,                     // Comma sign - ","
	                                         IN9 := #cs_PLCInfo,                // Message type - "PLCINFO"
	                                         IN10 := #cc_DL,                    // Comma sign - ","
	                                         IN11 := #ss_MsgID,                 // MSGID
	                                         IN12 := #cc_DL);                   // Comma sign - ","

	                    #ss_Message := CONCAT(IN1 := #ss_Speed,                 // Conveyor speed
	                                          IN2 := #cc_DL,                    // Comma sign - ","
	                                          IN3 := #ss_MachStat,              // Machine status
	                                          IN4 := #cc_DL,                    // Comma sign - ","
	                                          IN5 := #ss_SysRevs,               // System revolutions
	                                          IN6 := #cc_DL,                    // Comma sign - ","
	                                          IN7 := #ss_ActiveCamera,          // Active camera
	                                          IN8 := #cs_CRLF);                 // Termination signs - "$R$L"

	                    // Get the maximum number of the message array elements
	                    #si_MaxMsgLen := "FC_GetNrOfArrayEl"(iv_Array := #sUDT_MessageArray.Character);

	                    // Get the length of the complete message
	                    #si_MsgLen := LEN(#ss_Message) + LEN(#ss_Header);

	                    // Message array size validation
	                    #sa_Status.InvalidMsgArraySize := #si_MsgLen > #si_MaxMsgLen;

	                    // Convert header AND message charater strings into the message array OF characters
	                    IF (NOT #sa_Status.InvalidMsgArraySize)                 // Message character array size valid
	                    THEN

	                        Strg_TO_Chars(Strg := #ss_Header,                   // Convert message character string to Message character array
	                                      pChars := 0,
	                                      Cnt => #sui_ArrayOffset,
	                                      Chars := #sUDT_MessageArray.Character);

	                        Strg_TO_Chars(Strg := #ss_Message,                  // Convert message character string  to the char array
	                                      pChars := #sui_ArrayOffset,
	                                      Cnt => #sui_MsgArrayElNr,
	                                      Chars := #sUDT_MessageArray.Character);

	                    END_IF;

	                    // Clear remaining characters in message character array
	                    IF (NOT #sa_Status.InvalidMsgArraySize)                 // Message character array size is valid
	                    THEN

	                        // Filling up not used message character array elements with '$00' (ASCII - 16#00)
	                        FILL_BLK(IN := #cc_NULL,                            // Fill not used message char array elements with '$00'
	                                 COUNT := UINT_TO_ULINT(INT_TO_UINT(#si_MaxMsgLen) - #sui_MsgArrayElNr - #sui_ArrayOffset),
	                                 OUT => #sUDT_MessageArray.Character[#sui_MsgArrayElNr + #sui_ArrayOffset]);

	                    END_IF;

	                    // Move message into the FIFO buffer
	                    IF (NOT #sa_Status.InvalidMsgArraySize)                 // Message character array size is valid
	                    THEN

	                        // Mode 'W' - Write FIFO record
	                        "FC_Fifo"(ic_Mode := 'W',
	                                  qUDT_Status => #sa_Status.FIFOStatus,
	                                  qx_Error => #sa_Status.FIFOError,
	                                  qx_Warning => #sa_Status.FIFOWarning,
	                                  iqv_Data := #sUDT_MessageArray,
	                                  iqUDT_FifoHeader := #iqUDT_FifoHeader,
	                                  iqv_DataBuffer := #iqa_FifoData);


	                    END_IF;

	                    // In case of FIFO full, the FIFO full error bit and FIFO collective error bit are set
	                ELSE

	                    #sa_Status.FIFOError := TRUE;
	                    #sa_Status.FIFOStatus.FifoFull := TRUE;


	                END_IF;

	            END_IF;

	        END_REGION

	    END_IF;

	END_REGION

	REGION 3 – Status

	    // Create a collective error bit
	    #qx_Error :=
	    #sa_Status.InvalidSysRevs                   // Invalid system revolutions number
	    OR #sa_Status.InvalidSpeed                  // Invalid conveyor speed
	    OR #sa_Status.InvalidMsgArraySize           // Invalid message array size
	    OR #sa_Status.FIFOError;                    // FIFO error

	    // Create a collective warning bit
	    #qx_Warning := #sa_Status.FIFOWarning;      // FIFO warning

	END_REGION
END_FUNCTION_BLOCK

FUNCTION_BLOCK "FB_UPSSortConf"
TITLE = FB_SortConf
{ S7_Optimized_Access := 'TRUE' }
AUTHOR : MHSE
FAMILY : UPS_SpecificCommunication
VERSION : 3.0
// ATTRIBUTES
// AUTO_NUMBER = True
// BLOCK_NUMBER = 61
// END_ATTRIBUTES
//Function block to prepare and send the UPS SORTCONF message.
   VAR_INPUT
      iUDT_MsgHeader { ExternalAccessible := 'False'; ExternalVisible := 'False'; ExternalWritable := 'False'} : "UDT_UPSMessageHeader";   // UPS message header
      is_ActualDateTime { ExternalAccessible := 'False'; ExternalVisible := 'False'; ExternalWritable := 'False'} : String[23];   // Actual date and time
      is_ModuleName { ExternalAccessible := 'False'; ExternalVisible := 'False'; ExternalWritable := 'False'} : String[2] := 'AB';   // Module type
      is_DeviceNumber { ExternalAccessible := 'False'; ExternalVisible := 'False'; ExternalWritable := 'False'} : String[4] := 'abcd';   // Device number
      ii_GIN { ExternalAccessible := 'False'; ExternalVisible := 'False'; ExternalWritable := 'False'} : Int;   // GIN
      ii_Destination { ExternalAccessible := 'False'; ExternalVisible := 'False'; ExternalWritable := 'False'} : Int;   // Chute destination
      ii_GINRangeStart { ExternalAccessible := 'False'; ExternalVisible := 'False'; ExternalWritable := 'False'} : Int;   // Valid GIN range start
      ii_GINRangeEnd { ExternalAccessible := 'False'; ExternalVisible := 'False'; ExternalWritable := 'False'} : Int;   // Valid GIN range end
   END_VAR

   VAR_OUTPUT
      qx_Error { ExternalAccessible := 'False'; ExternalVisible := 'False'; ExternalWritable := 'False'} : Bool;   // Collective error output
      qx_Warning { ExternalAccessible := 'False'; ExternalVisible := 'False'; ExternalWritable := 'False'} : Bool;   // Collective warning output
   END_VAR

   VAR_IN_OUT
      iqUDT_EquipmentControl : "UDT_EquipmentControl";   // Equipment control structure
      iqUDT_LostStatistics : "UDT_UPSLostCounters";   // Lost parcels statistics
      iqUDT_FifoHeader : "UDT_FifoHeader";   // FIFO header
      iqa_FifoData : Array[*] of "UDT_Message";   // FIFO data
      iqdi_UniqueMsgID { ExternalAccessible := 'False'; ExternalVisible := 'False'; ExternalWritable := 'False'} : DInt;   // Unique message ID integer
   END_VAR

   VAR
      sUDT_MessageArray { ExternalAccessible := 'False'; ExternalVisible := 'False'; ExternalWritable := 'False'; S7_SetPoint := 'False'} : "UDT_Message";   // Message character array
      ss_Status { ExternalAccessible := 'False'; ExternalVisible := 'False'; ExternalWritable := 'False'} : Struct   // Status structure
         FIFOStatus { ExternalAccessible := 'False'; ExternalVisible := 'False'; ExternalWritable := 'False'} : "UDT_FifoStatus";   //  FIFO status structure
         FIFOError { ExternalAccessible := 'False'; ExternalVisible := 'False'; ExternalWritable := 'False'; S7_SetPoint := 'True'} : Bool;   //  FIFO error
         FIFOWarning { ExternalAccessible := 'False'; ExternalVisible := 'False'; ExternalWritable := 'False'; S7_SetPoint := 'True'} : Bool;   //  FIFO warning
         InvalidPkgRevs { ExternalAccessible := 'False'; ExternalVisible := 'False'; ExternalWritable := 'False'} : Bool;   //  Invalid package revolutions number
         InvalidGIN { ExternalAccessible := 'False'; ExternalVisible := 'False'; ExternalWritable := 'False'} : Bool;   //  Invalid GIN
         InvalidDest { ExternalAccessible := 'False'; ExternalVisible := 'False'; ExternalWritable := 'False'} : Bool;   //  Invalid destination
         InvalidMsgArraySize { ExternalAccessible := 'False'; ExternalVisible := 'False'; ExternalWritable := 'False'} : Bool;   //  Invalid message array size
      END_STRUCT;
      sa_PKGSTATArray { ExternalAccessible := 'False'; ExternalVisible := 'False'; ExternalWritable := 'False'} : Array[0..4] of Byte;   // PKGSTAT
      ss_Dest { ExternalAccessible := 'False'; ExternalVisible := 'False'; ExternalWritable := 'False'} : String[5];   // Destination
      ss_PACKREVS { ExternalAccessible := 'False'; ExternalVisible := 'False'; ExternalWritable := 'False'} : String[4];   // Package revolutions
      ss_Message { ExternalAccessible := 'False'; ExternalVisible := 'False'; ExternalWritable := 'False'} : String;   // Message character string
      ss_PKGSTAT { ExternalAccessible := 'False'; ExternalVisible := 'False'; ExternalWritable := 'False'} : String;   // Message delay
      ss_PKGSTATPart { ExternalAccessible := 'False'; ExternalVisible := 'False'; ExternalWritable := 'False'} : String;   // Message delay
      sui_MsgArrayElNr { ExternalAccessible := 'False'; ExternalVisible := 'False'; ExternalWritable := 'False'} : UInt;   // Number of written message characters
      si_MaxMsgLen { ExternalAccessible := 'False'; ExternalVisible := 'False'; ExternalWritable := 'False'} : Int;   // Maximum message length
      si_MsgLen { ExternalAccessible := 'False'; ExternalVisible := 'False'; ExternalWritable := 'False'} : Int;   // String character message length
      si_GINLen { ExternalAccessible := 'False'; ExternalVisible := 'False'; ExternalWritable := 'False'} : Int;   // GIN array length
      si_PACKREVSLen { ExternalAccessible := 'False'; ExternalVisible := 'False'; ExternalWritable := 'False'} : Int;   // Package revolutions string length
      si_DestLen { ExternalAccessible := 'False'; ExternalVisible := 'False'; ExternalWritable := 'False'} : Int;   // Destination string length
      si_i { ExternalAccessible := 'False'; ExternalVisible := 'False'; ExternalWritable := 'False'} : Int;   // Loop counter
   END_VAR
   VAR RETAIN
      si_OldGIN { ExternalAccessible := 'False'; ExternalVisible := 'False'; ExternalWritable := 'False'} : Int;   // Old GIN
   END_VAR

   VAR CONSTANT
      cc_NULL : Char := '$00';   // NULL sign
      cc_DL : Char := ',';   // Comma sign
      cc_Dash : Char := '-';   // Dash sign
      cs_CRLF : String := '$R$L';   // Termination signs
      cs_SortConf : String := 'SORTCONF';   // Message type
   END_VAR


BEGIN
	(*
	----------------------------------------------------------------------------------------

	Version history:
	Date        | Version   | Author        | Remark
	----------------------------------------------------------------------------------------
	24/05/2019  | 0.1       | L.Klar        | first release MHS TIA 15.1
	13/06/2019  | 0.2       | A.Nowak       | Replacement of instruction if for direct write into variable - Region 3 and 4 and 5 and 6.8 , changing and for or in conditions in regions 3 and 4 and 5
	28/06/2019  | 0.4       | A.Nowak       | Changing conditions for error occuring and status update
	18/07/2019  | 0.5       | L.Klar        | Status handling changed
	24/07/2019  | 2.0       | L.Klar        | 2.0 MHS library release TIA 15.1
	23/08/2019  | 2.1       | K.Pokorski    | Bool to byte block changed to direct reference, comments simplified
	20/09/2019  | 2.2       | M.Kurpiers    | Change - status to struct
	01/10/2019  | 2.3       | A.Nowak       | Implementation of the new FIFO block
	12/11/2019  | 3.0       | P.Majka       | 3.0 MHS library release TIA 15.1
	09/01/2020  | 3.1       | L.Klar        | Parcel status handling changed
	01/10/2020  | 3.2       | L.Klar        | Invalid package revolution error condition changed to handle 0
	                                        | Message trigger based on new GIN detection
	14/12/2020  | 3.3       | L.Klar        | ID created bit changed, destination too late reset if no detination received
	14/12/2020  | 3.4       | L.Klar        | Statistics for BAU added
	22/02/2023  | 4.0       | F.Baten       | 4.0 Release TIA 17.5
	02/05/2024  | 4.1       | J.Majer      | Datatype conversions changed from automatic to explicit, to accomodate IEC 61131-3 standard
	*)

	REGION 1 - Reset statistics

	    IF #iqUDT_EquipmentControl.Command.ResetData THEN

	        #iqUDT_LostStatistics.LostInTracking := 0;
	        #iqUDT_LostStatistics.NoUPSID := 0;
	        #iqUDT_LostStatistics.NoSortRcv := 0;

	    END_IF;

	END_REGION

	REGION 2 – SortConf

	    IF #ii_GIN <> #si_OldGIN
	        AND #ii_GIN >= #ii_GINRangeStart
	        AND #ii_GIN <= #ii_GINRangeEnd
	    THEN

	        #si_OldGIN := #ii_GIN;

	        REGION 2.1 – Update the FIFO header status bits

	            // Mode 'S' - FIFO register status update
	            "FC_Fifo"(ic_Mode := 'S',
	                      qUDT_Status => #ss_Status.FIFOStatus,
	                      qx_Error => #ss_Status.FIFOError,
	                      qx_Warning => #ss_Status.FIFOWarning,
	                      iqv_Data := #sUDT_MessageArray,
	                      iqUDT_FifoHeader := #iqUDT_FifoHeader,
	                      iqv_DataBuffer := #iqa_FifoData);


	        END_REGION

	        REGION 2.2 – Maximum number of the package information's array elements

	            #si_GINLen := "FC_GetNrOfArrayEl"(iv_Array := "DB_GIN".GIN);

	        END_REGION

	        REGION 2.3 – GIN validation

	            #ss_Status.InvalidGIN :=
	            #ii_GIN <= 0
	            OR #ii_GIN > #si_GINLen;

	        END_REGION

	        REGION 2.4 – Number of recirculations validation

	            IF (NOT #ss_Status.InvalidGIN)
	            THEN

	                #ss_Status.InvalidPkgRevs :=
	                "DB_GIN".GIN[#ii_GIN].General.NrOfRecirculations < 0
	                OR "DB_GIN".GIN[#ii_GIN].General.NrOfRecirculations > 9999;

	            END_IF;

	        END_REGION

	        REGION 2.5 – Destination validation

	            IF (NOT #ss_Status.InvalidGIN)
	            THEN

	                #ss_Status.InvalidDest :=
	                "DB_GIN".GIN[#ii_GIN].General.Destination[0] < 0
	                OR "DB_GIN".GIN[#ii_GIN].General.Destination[0] >= 10000;

	            END_IF;

	        END_REGION

	        REGION 2.6 - Sort statistics

	            IF "DB_GIN".GIN[#ii_GIN].General.DestRcv THEN
	                "DB_GIN".GIN[#ii_GIN].UPS.IDCreated := TRUE;
	            END_IF;

	            IF NOT "DB_GIN".GIN[#ii_GIN].General.Lost THEN
	                IF "DB_GIN".GIN[#ii_GIN].UPS.IDCreated THEN
	                    IF NOT "DB_GIN".GIN[#ii_GIN].General.DestRcv THEN
	                        #iqUDT_LostStatistics.NoSortRcv += 1;
	                    END_IF;
	                ELSE
	                    #iqUDT_LostStatistics.NoUPSID += 1;
	                END_IF;
	            ELSE
	                #iqUDT_LostStatistics.LostInTracking += 1;
	            END_IF;

	        END_REGION

	        REGION 2.7 – SORTCONF message preparation

	            // Conditions of sending the message
	            IF (NOT #ss_Status.FIFOError
	                AND NOT #ss_Status.InvalidGIN
	                AND NOT #ss_Status.InvalidPkgRevs
	                AND NOT #ss_Status.InvalidDest)
	            THEN

	                IF (NOT #iqUDT_FifoHeader.Status.Full)
	                THEN

	                    // Unique  MSGID
	                    "FC_UPSMsgId"(is_ActualDateTime := #is_ActualDateTime,
	                                  is_ModuleName := #is_ModuleName,
	                                  is_DeviceNumber := #is_DeviceNumber,
	                                  iqs_MSGID := "DB_GIN".GIN[#ii_GIN].UPS.MSGID,
	                                  iqdi_UniqueMsgID := #iqdi_UniqueMsgID);

	                    // Sort status

	                    // Parcel diverted
	                    "DB_GIN".GIN[#ii_GIN].General.SortStatus.NoDivert := FALSE;

	                    // Good divert
	                    "DB_GIN".GIN[#ii_GIN].General.SortStatus.GoodDivert := #ii_Destination = "DB_GIN".GIN[#ii_GIN].General.Destination[0] AND NOT "DB_GIN".GIN[#ii_GIN].General.Lost;

	                    // Divert failed
	                    "DB_GIN".GIN[#ii_GIN].General.SortStatus.FailedDivert := NOT "DB_GIN".GIN[#ii_GIN].General.SortStatus.GoodDivert;

	                    "DB_GIN".GIN[#ii_GIN].General.SortStatus.DivertDestination := #ii_Destination;


	                    IF "DB_GIN".GIN[#ii_GIN].General.SortStatus.FailedDivert
	                    THEN
	                        IF NOT "DB_GIN".GIN[#ii_GIN].General.Lost THEN
	                            "DB_GIN".GIN[#ii_GIN].General.SortStatus.NoDivertCause.NoDestRcv := NOT "DB_GIN".GIN[#ii_GIN].General.DestRcv;
	                            "DB_GIN".GIN[#ii_GIN].General.SortStatus.NoDivertCause.DestTooLate := "DB_GIN".GIN[#ii_GIN].General.DestRcv;
	                        ELSE
	                            "DB_GIN".GIN[#ii_GIN].General.SortStatus.NoDivertCause.NoDestRcv := FALSE;
	                            "DB_GIN".GIN[#ii_GIN].General.SortStatus.NoDivertCause.DestTooLate := FALSE;
	                        END_IF;
	                    END_IF;

	                    // Package status - PKGSTAT2

	                    #sa_PKGSTATArray[0].%X0 := "DB_GIN".GIN[#ii_GIN].UPS.IDCreated;                                         // Byte 1, Bit 0 - PLCID created or TrayID Read (Package Passed through Camera Tunnel
	                    #sa_PKGSTATArray[0].%X1 := "DB_GIN".GIN[#ii_GIN].UPS.DimDataRcv;                                        // Byte 1, Bit 1 - Package Dimensional Data Received via Camera Scan Data Message
	                    #sa_PKGSTATArray[0].%X2 := "DB_GIN".GIN[#ii_GIN].UPS.PkgWrongInduct;                                    // Byte 1, Bit 2 - Package Did NOT Induct Properly (Non-Tray Systems)
	                    #sa_PKGSTATArray[0].%X3 := "DB_GIN".GIN[#ii_GIN].General.DestRcv;                                       // Byte 1, Bit 3 - SORT Command Received
	                    #sa_PKGSTATArray[0].%X4 := "DB_GIN".GIN[#ii_GIN].General.SortStatus.NoDivertCause.DestTooLate;          // Byte 1, Bit 4 - SORT Command Late
	                    #sa_PKGSTATArray[0].%X5 := "DB_GIN".GIN[#ii_GIN].General.SortStatus.NoDivertCause.InvalidDest;          // Byte 1, Bit 5 - SORT Command Invalid Destination
	                    #sa_PKGSTATArray[0].%X6 := "DB_GIN".GIN[#ii_GIN].General.SortStatus.NoDivertCause.NoDestRcv;            // Byte 1, Bit 6 - No SORT message Received for PKG or TRAY ID
	                    #sa_PKGSTATArray[0].%X7 := "DB_GIN".GIN[#ii_GIN].General.SortStatus.GoodDivert;                         // Byte 1, Bit 7 - Good Divert / Sort


	                    #sa_PKGSTATArray[1].%X0 := "DB_GIN".GIN[#ii_GIN].UPS.IDCalcFromCamID;                                   // Byte 2, Bit 0 - PLCID/TrayID Calculated From CamID
	                    #sa_PKGSTATArray[1].%X1 := "DB_GIN".GIN[#ii_GIN].General.SortStatus.NoDivert;                           // Byte 2, Bit 1 - Divert/Tip Attempted
	                    #sa_PKGSTATArray[1].%X2 := "DB_GIN".GIN[#ii_GIN].General.SortStatus.NoDivertCause.TrayDisabled;         // Byte 2, Bit 2 - Tray Disabled (Tray Systems)
	                    #sa_PKGSTATArray[1].%X3 := "DB_GIN".GIN[#ii_GIN].General.SortStatus.NoDivertCause.DestDisabled;         // Byte 2, Bit 3 - Destination Disabled (via HMI or PFC)
	                    #sa_PKGSTATArray[1].%X4 := "DB_GIN".GIN[#ii_GIN].UPS.UnknownParcelID;                                   // Byte 2, Bit 4 - Unknown Parcel ID
	                    #sa_PKGSTATArray[1].%X5 := "DB_GIN".GIN[#ii_GIN].UPS.UndefinedProblem;                                  // Byte 2, Bit 5 - Un-Defined Problem
	                    #sa_PKGSTATArray[1].%X6 := "DB_GIN".GIN[#ii_GIN].UPS.UnrecognizedCmd;                                   // Byte 2, Bit 6 - Un-recognized command
	                    #sa_PKGSTATArray[1].%X7 := "DB_GIN".GIN[#ii_GIN].UPS.SorterInMainteneceMode;                            // Byte 2, Bit 7 - Sorter in Maintenance/Commissioning Mode


	                    #sa_PKGSTATArray[2].%X0 := "DB_GIN".GIN[#ii_GIN].General.SortStatus.NoDivertCause.ChuteJam;             // Byte 3, Bit 0 - Chute Jam
	                    #sa_PKGSTATArray[2].%X1 := "DB_GIN".GIN[#ii_GIN].General.SortStatus.FailedDivert;                       // Byte 3, Bit 1 - Failed Divert
	                    #sa_PKGSTATArray[2].%X2 := "DB_GIN".GIN[#ii_GIN].General.Lost;                                          // Byte 3, Bit 2 - Parcel Lost in PFC Tracking
	                    #sa_PKGSTATArray[2].%X3 := "DB_GIN".GIN[#ii_GIN].UPS.DestUserSusp;                                      // Byte 3, Bit 3 - Destination User Suspended
	                    #sa_PKGSTATArray[2].%X4 := "DB_GIN".GIN[#ii_GIN].General.SortStatus.NoDivertCause.ChuteFull;            // Byte 3, Bit 4 - Chute Full / Bag Closed
	                    #sa_PKGSTATArray[2].%X5 := "DB_GIN".GIN[#ii_GIN].General.SortStatus.NoDivertCause.SorterNotAtSpeed;     // Byte 3, Bit 5 - Sorter NOT At Speed
	                    #sa_PKGSTATArray[2].%X6 := "DB_GIN".GIN[#ii_GIN].UPS.SorterNotSynch;                                    // Byte 3, Bit 6 - Sorter NOT Synchronized (Tilt Tray Systems)
	                    #sa_PKGSTATArray[2].%X7 := FALSE;                                                                       // Byte 3, Bit 7 - Max Recirculation (Revolving Systems)


	                    #sa_PKGSTATArray[3].%X0 := "DB_GIN".GIN[#ii_GIN].UPS.PkgDetAtVerCheckPoint;                             // Byte 4, Bit 0 - Package Detected at Verification Check Point
	                    #sa_PKGSTATArray[3].%X1 := "DB_GIN".GIN[#ii_GIN].General.SortStatus.NoDivertCause.LeadingGapError;      // Byte 4, Bit 1 - Gap Error Leading Edge
	                    #sa_PKGSTATArray[3].%X2 := "DB_GIN".GIN[#ii_GIN].General.SortStatus.NoDivertCause.TrailingGapError;     // Byte 4, Bit 2 - Gap Error Trailing Edge
	                    #sa_PKGSTATArray[3].%X3 := "DB_GIN".GIN[#ii_GIN].General.PkgTooHigh;                                    // Byte 4, Bit 3 - Package Too Tall
	                    #sa_PKGSTATArray[3].%X4 := "DB_GIN".GIN[#ii_GIN].General.PkgTooSmall;                                   // Byte 4, Bit 4 - Package Too Small
	                    #sa_PKGSTATArray[3].%X5 := "DB_GIN".GIN[#ii_GIN].General.PkgTooLong;                                    // Byte 4, Bit 5 - Package Too Long
	                    #sa_PKGSTATArray[3].%X6 := "DB_GIN".GIN[#ii_GIN].General.SortStatus.NoDivertCause.DestNotReachable;     // Byte 4, Bit 6 - Crossover Destination
	                    #sa_PKGSTATArray[3].%X7 := "DB_GIN".GIN[#ii_GIN].UPS.ChuteFullAftrAlterDest;                            // Byte 4, Bit 7 - Preferred chute full after passed alternate destination


	                    #sa_PKGSTATArray[4].%X0 := "DB_GIN".GIN[#ii_GIN].UPS.ChuteNotAvailAfterAlterDest;                       // Byte 5, Bit 0 - Preferred chute not available after passed alternate destination
	                    #sa_PKGSTATArray[4].%X1 := "DB_GIN".GIN[#ii_GIN].General.SortStatus.NoDivertCause.NoRTR;                // Byte 5, Bit 1 - Take away conveyor not running
	                    #sa_PKGSTATArray[4].%X2 := "DB_GIN".GIN[#ii_GIN].UPS.PLCRedirected;                                     // Byte 5, Bit 2 - PLC Redirected
	                    #sa_PKGSTATArray[4].%X3 := FALSE;                                                                       // Byte 5, Bit 3 - Future / or Machine Specific (To be identified)
	                    #sa_PKGSTATArray[4].%X4 := FALSE;                                                                       // Byte 5, Bit 4 - Future / or Machine Specific (To be identified)
	                    #sa_PKGSTATArray[4].%X5 := FALSE;                                                                       // Byte 5, Bit 5 - Future / or Machine Specific (To be identified)
	                    #sa_PKGSTATArray[4].%X6 := FALSE;                                                                       // Byte 5, Bit 6 - Future / or Machine Specific (To be identified)
	                    #sa_PKGSTATArray[4].%X7 := FALSE;                                                                       // Byte 5, Bit 7 - Future / or Machine Specific (To be identified)

	                    // PKGSTAT character string clearing
	                    #ss_PKGSTAT := '';

	                    // PKGSTAT bytes conversion to character string
	                    FOR #si_i := 0 TO 4 DO

	                        // Initialize the part of the PKGSTAT character string
	                        #ss_PKGSTATPart := '';

	                        // PKGSTAT byte conversion to string
	                        VAL_STRG(IN := BYTE_TO_USINT(#sa_PKGSTATArray[#si_i]),
	                                 SIZE := 0,
	                                 PREC := 0,
	                                 FORMAT := 0,
	                                 P := 1,
	                                 OUT => #ss_PKGSTATPart);

	                        // PKGSTAT character string building
	                        IF (#si_i < 4)              // Loop counter lower than 4
	                        THEN

	                            #ss_PKGSTAT := CONCAT(IN1 := #ss_PKGSTAT,
	                                                  IN2 := #ss_PKGSTATPart,
	                                                  IN3 := #cc_Dash);

	                        ELSE

	                            #ss_PKGSTAT := CONCAT(IN1 := #ss_PKGSTAT,
	                                                  IN2 := #ss_PKGSTATPart);
	                        END_IF;

	                    END_FOR;

	                    // Package revolutions - PACKREVS

	                    // Package revolutions number character string clearing
	                    #ss_PACKREVS := '';

	                    // Package revolutions number integer converion to a character string
	                    VAL_STRG(IN := "DB_GIN".GIN[#ii_GIN].General.NrOfRecirculations,
	                             SIZE := 0,
	                             PREC := 0,
	                             FORMAT := 0,
	                             P := 1,
	                             OUT => #ss_PACKREVS);

	                    // Length of the package revolutions number character string
	                    #si_PACKREVSLen := LEN(#ss_PACKREVS);

	                    // Package revolutions number character string leading zeros addition
	                    IF (#si_PACKREVSLen < 4)        // Package revolutions string length is lower than 4
	                    THEN

	                        FOR #si_i := 1 TO 4 - #si_PACKREVSLen DO

	                            #ss_PACKREVS := CONCAT(IN1 := '0',
	                                                   IN2 := #ss_PACKREVS);

	                        END_FOR;

	                    END_IF;

	                    // Destination - DEST

	                    // Initialize the destination character String
	                    #ss_Dest := '';

	                    // Destionation value integer converion to a character string
	                    VAL_STRG(IN := "DB_GIN".GIN[#ii_GIN].General.SortStatus.DivertDestination,
	                             SIZE := 0,
	                             PREC := 0,
	                             FORMAT := 0,
	                             P := 1,
	                             OUT => #ss_Dest);

	                    // Length of the destination character string
	                    #si_DestLen := LEN(#ss_Dest);

	                    // Destination character string leading zeros addition
	                    IF (#si_DestLen < 5)        // Destination string length
	                    THEN

	                        FOR #si_i := 1 TO 5 - #si_DestLen DO

	                            #ss_Dest := CONCAT(IN1 := '0',
	                                               IN2 := #ss_Dest);

	                        END_FOR;

	                    END_IF;

	                    // Message preparation

	                    // SORTCANF message composing according to the structure: SCN,SCT,RCN,RCT,MT,PKGUID,TRKNUM,Dest,PKGSTAT,PACKREVS {CRLF}
	                    #ss_Message := CONCAT(IN1 := #iUDT_MsgHeader.SCN,                  // Sender IP address
	                                          IN2 := #cc_DL,                                // Comma sign - ","
	                                          IN3 := #iUDT_MsgHeader.SCT,                  // Sender Name
	                                          IN4 := #cc_DL,                                // Comma sign - ","
	                                          IN5 := #iUDT_MsgHeader.RCN,                  // Receiver IP address
	                                          IN6 := #cc_DL,                                // Comma sign - ","
	                                          IN7 := #iUDT_MsgHeader.RCT,                  // Receiver Name)
	                                          IN8 := #cc_DL,                                // Comma sign - ","
	                                          IN9 := #cs_SortConf,                          // Message type - "SORTCONF"
	                                          IN10 := #cc_DL,                               // Comma sign - ","
	                                          IN11 := "DB_GIN".GIN[#ii_GIN].UPS.MSGID,      // MSGID
	                                          IN12 := #cc_DL,                               // Comma sign - ","
	                                          IN13 := "DB_GIN".GIN[#ii_GIN].UPS.PKGUID,     // Package unique ID
	                                          IN14 := #cc_DL,                               // Comma sign - ","
	                                          IN15 := "DB_GIN".GIN[#ii_GIN].UPS.TRKNUM,     // Tracking number
	                                          IN16 := #cc_DL,                               // Comma sign - ","
	                                          IN17 := #ss_Dest,                             // Destination
	                                          IN18 := #cc_DL,                               // Comma sign - ","
	                                          IN19 := #ss_PKGSTAT,                          // Package status
	                                          IN20 := #cc_DL,                               // Comma sign - ","
	                                          IN21 := #ss_PACKREVS,                         // Package revolutions
	                                          IN22 := #cs_CRLF);                            // Termination signs - "$R$L"

	                    // Maximum number of the message characters
	                    #si_MaxMsgLen := "FC_GetNrOfArrayEl"(iv_Array := #sUDT_MessageArray.Character);

	                    // Length of the complete message
	                    #si_MsgLen := LEN(#ss_Message);

	                    // Message array size validation
	                    #ss_Status.InvalidMsgArraySize := #si_MsgLen > #si_MaxMsgLen;

	                    // Message charater string conversion to a Message array characters
	                    IF (NOT #ss_Status.InvalidMsgArraySize)
	                    THEN

	                        Strg_TO_Chars(Strg := #ss_Message,
	                                      pChars := 0,
	                                      Cnt => #sui_MsgArrayElNr,
	                                      Chars := #sUDT_MessageArray.Character);

	                    END_IF;

	                    // Clearing remaining characters in message character array
	                    IF (NOT #ss_Status.InvalidMsgArraySize)
	                    THEN

	                        // Filling up not used message character array elements with '$00' (ASCII - 16#00)
	                        FILL_BLK(IN := #cc_NULL,
	                                 COUNT := UINT_TO_ULINT(INT_TO_UINT(#si_MaxMsgLen) - #sui_MsgArrayElNr),
	                                 OUT => #sUDT_MessageArray.Character[#sui_MsgArrayElNr]);

	                    END_IF;

	                    // Message write into a FIFO register
	                    IF (NOT #ss_Status.InvalidMsgArraySize)

	                    THEN

	                        // Mode 'W' - Write FIFO record
	                        "FC_Fifo"(ic_Mode := 'W',
	                                  qUDT_Status => #ss_Status.FIFOStatus,
	                                  qx_Error => #ss_Status.FIFOError,
	                                  qx_Warning => #ss_Status.FIFOWarning,
	                                  iqv_Data := #sUDT_MessageArray,
	                                  iqUDT_FifoHeader := #iqUDT_FifoHeader,
	                                  iqv_DataBuffer := #iqa_FifoData);


	                    END_IF;

	                    // In case of FIFO full, the FIFO full error bit and FIFO collective error bit are set
	                ELSE

	                    #ss_Status.FIFOError := TRUE;
	                    #ss_Status.FIFOStatus.FifoFull := TRUE;

	                END_IF;

	            END_IF;

	        END_REGION

	        REGION 2.8 – Status

	            // Create a collective error bit
	            #qx_Error :=
	            #ss_Status.InvalidDest
	            OR #ss_Status.InvalidPkgRevs
	            OR #ss_Status.InvalidGIN
	            OR #ss_Status.InvalidMsgArraySize
	            OR #ss_Status.FIFOError;

	            // Create a collective warning bit
	            #qx_Warning := #ss_Status.FIFOWarning;

	        END_REGION

	    END_IF;

	END_REGION
END_FUNCTION_BLOCK

FUNCTION_BLOCK "FB_UPSSafetyZoneStatistics"
{ S7_Optimized_Access := 'TRUE' }
VERSION : 0.1
// ATTRIBUTES
// AUTO_NUMBER = True
// BLOCK_NUMBER = 60
// END_ATTRIBUTES
   VAR_INPUT
      iUDT_EquipmentControl { ExternalAccessible := 'False'; ExternalVisible := 'False'; ExternalWritable := 'False'} : "UDT_EquipmentControl";   // Equipment control structure
      ix_SafetyZoneOK { ExternalAccessible := 'False'; ExternalVisible := 'False'; ExternalWritable := 'False'} : Bool;   // SSP Field input
   END_VAR

   VAR_OUTPUT
      qx_SafetyZoneOK { ExternalAccessible := 'False'; ExternalVisible := 'False'; ExternalWritable := 'False'} : Bool;
   END_VAR

   VAR_IN_OUT
      iqUDT_Statistics : "UDT_UPSSafetyZoneStatistics";
   END_VAR

   VAR
      sR_TRIG_NotHealthy {InstructionName := 'R_TRIG'; LibVersion := '1.0'; ExternalAccessible := 'False'; ExternalVisible := 'False'; ExternalWritable := 'False'; S7_SetPoint := 'False'} : R_TRIG;   // Rising edge start
      sx_safetyZoneOk { ExternalAccessible := 'False'; ExternalVisible := 'False'; ExternalWritable := 'False'} : Bool;
   END_VAR


BEGIN
	(*
	----------------------------------------------------------------------------------------

	Version history:
	Date        | Version   | Author        | Remark
	----------------------------------------------------------------------------------------
	17/08/2020  | 1.0       | S. Theocharis | First release
	22/02/2023  | 4.0       | F.Baten       | 4.0 Release TIA 17.5
	*)


	REGION 1 Safety Zone ok mapping

	    #qx_SafetyZoneOK := #sx_safetyZoneOk := #ix_SafetyZoneOK;

	END_REGION


	REGION 2 Statistics

	    REGION 2.1 Trigger
	        //Start trigger
	        #sR_TRIG_NotHealthy(CLK := NOT #sx_safetyZoneOk);

	    END_REGION

	    REGION 2.2 Not Healthy

	        IF (NOT #sx_safetyZoneOk
	            OR #iUDT_EquipmentControl.Command.ResetData)                                          // Reset statistics
	        THEN

